FUNCTION_BLOCK FB_Clamp01_Test EXTENDS TcUnit.FB_TestSuite

TestCase('Value Limit Min Overflow', fValue := -0.1, fExpected:= 0);
TestCase('Value Limit Min',fValue := 0.0, fExpected:= 0);
TestCase('Value In Range ',fValue := 0.5, fExpected:= 0.5);
TestCase('Value Limit Max',fValue := 1, fExpected:= 1);
TestCase('Value Limit Max Overflow',fValue := 1.1, fExpected:= 1);

METHOD TestCase
VAR_INPUT
	sName : T_MaxString;
	fValue : REAL;
	fExpected : REAL;
END_VAR

VAR	
	fResult : REAL;
END_VAR
TEST(sName);
	
fResult := F_Clamp01(fValue);
AssertEquals(Expected := fExpected,
             Actual := fResult,
             Message := 'Result value is not correct');	
	 
TEST_FINISHED();
END_METHOD

END_FUNCTION_BLOCK

(* stored: Version 1.1.0.1, ProductVersion 3.1.4024.12
   POU FB_Clamp01_Test: Id {25fbacd2-212e-077a-2ecf-41abb0aa3aa3}, SpecialFunc None
   Method TestCase: Id {99da69e4-852b-0a97-230b-10782ad258b3} *)
